# EPICS autosave request: support/ebrick/2-2-3/iocBoot/iocebrick/autosave/ebrickBITinp.req
$(P)$(H)$(F)$(D).SCAN
$(P)$(H)$(F)$(D).ZNAM
$(P)$(H)$(F)$(D).ONAM
$(P)$(H)$(F)$(D).DESC
